{attribute 'GeneratedUsingTerminal: EL2642-0000-0016'}
{attribute addProperty BoxType "EL2642-0000-0016"}
{attribute addProperty Id "DO_Inputs_DeviceAT %I*DO_Inputs_Device_4A9049C53DO_Group_1_OutputsAT %Q*DO_Group_1_Outputs_59D8C01C4DO_Group_2_OutputsAT %Q*DO_Group_2_Outputs_828082884WcStateAT %I*WcState_9091E0EB2InfoDataAT %I*InfoData_1088C70510"}
{attribute addProperty CRC "1285670039"}
{attribute addProperty Size "23"}
TYPE EL2642_4CA1C497 EXTENDS EtcSlaveTerminalBase_947E5A46 :
STRUCT
	{attribute addProperty Name "DO_Inputs_Device"}
	DO_Inputs_Device : DO_Inputs_Device_4A9049C5;
	{attribute addProperty Name "DO_Group_1_Outputs"}
	DO_Group_1_Outputs : DO_Group_1_Outputs_59D8C01C;
	{attribute addProperty Name "DO_Group_2_Outputs"}
	DO_Group_2_Outputs : DO_Group_2_Outputs_82808288;
	{attribute addProperty Name "WcState"}
	WcState : WcState_9091E0EB;
	{attribute addProperty Name "InfoData"}
	InfoData : InfoData_1088C705;
END_STRUCT
END_TYPE

(* stored: Version 1.2.0.0, ProductVersion 3.1.4024.9
   DUT EL2642_4CA1C497: Id {c862722f-1912-4cf6-954f-c3b601b04cb6} *)
